FUNCTION_BLOCK F_EXPT (* exponentiation *)
  (* Standard: 61131-3; Classification: standard arithmetic function; Description: Copyright (c) 2013 TU Wien ACIN This program and the accompanying materials are made available under the terms of the Eclipse Public License 2.0 which is available at https://www.eclipse.org/legal/epl-2.0/ SPDX-License-Identifier: EPL-2.0 *)
  (* Version 1.0, 2013-08-17, Monika Wenger, TU Wien ACIN *)
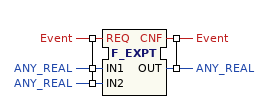
  EVENT_INPUT
    REQ WITH IN1, IN2; (* Normal Execution Request *)
  END_EVENT
  EVENT_OUTPUT
    CNF WITH OUT; (* Execution Confirmation *)
  END_EVENT
  VAR_INPUT
    IN1 : ANY_REAL; (* base input *)
    IN2 : ANY_REAL; (* exponent input *)
  END_VAR
  VAR_OUTPUT
    OUT : ANY_REAL; (* Function output *)
  END_VAR
END_FUNCTION_BLOCK
